FUNCTION_BLOCK Tank_Interface (* Composite FB wrapping other FBs *)
  (* Standard: 61499-2 *)
  (* Version 1.0, 2025-12-25, guilh *)
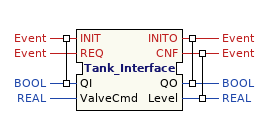
  EVENT_INPUT
    INIT WITH QI; (* Initialization Request *)
    REQ; (* Normal Execution Request *)
  END_EVENT
  EVENT_OUTPUT
    INITO WITH QO; (* Initialization Confirm *)
    CNF WITH Level; (* Execution Confirmation *)
  END_EVENT
  VAR_INPUT
    QI : BOOL; (* Input event qualifier *)
    ValveCmd : REAL;
  END_VAR
  VAR_OUTPUT
    QO : BOOL; (* Output event qualifier *)
    Level : REAL;
  END_VAR
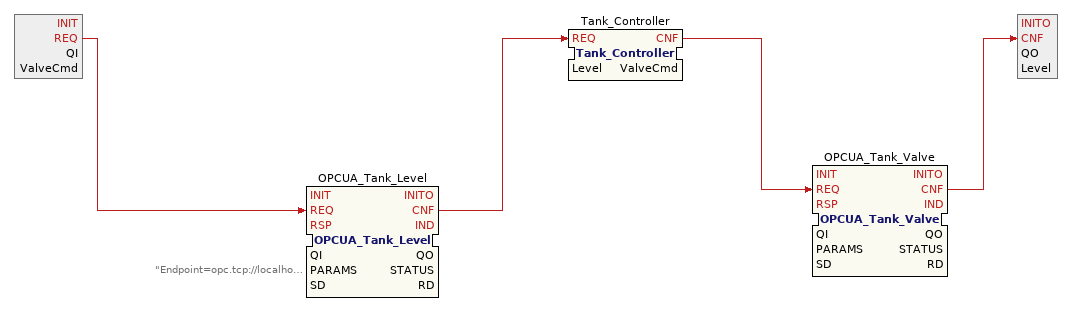
  FBS
    OPCUA_Tank_Level : OPCUA_Tank_Level(PARAMS := "Endpoint=opc.tcp://localhost:4840/freeopcua/server/;NodeId=ns=2;s=Tank.Level;Type=REAL;");
    Tank_Controller : Tank_Controller;
    OPCUA_Tank_Valve : OPCUA_Tank_Valve;
  END_FBS
  EVENT_CONNECTIONS
    REQ TO OPCUA_Tank_Level.REQ;
    OPCUA_Tank_Level.CNF TO Tank_Controller.REQ;
    Tank_Controller.CNF TO OPCUA_Tank_Valve.REQ;
    OPCUA_Tank_Valve.CNF TO CNF;
  END_CONNECTIONS
END_FUNCTION_BLOCK
